PROGRAM Watering
VAR
END_VAR

END_PROGRAM

(* stored: Version 1.1.0.1, ProductVersion 3.1.4024.15
   POU Watering: Id {3c8812c0-276c-4c26-8d31-84af572d2303}, SpecialFunc None *)
